// TIA Portal V17 export
// export: Created 2025-05-06T14:32:49.8619923Z, ExportSetting WithDefaults, DisplayName Totally Integrated Automation Portal, DisplayVersion V17 Update 8, DisplayName TIA Portal Openness, DisplayVersion V17 Update 8, DisplayName TIA Portal Version Control Interface, DisplayVersion V17, DisplayName SINAMICS Startdrive Advanced, DisplayVersion V17 SP2, DisplayName SINAMICS Startdrive G110M, G120, G120C, G120D, G120P, G115D, DisplayVersion V17 SP2, DisplayName SINAMICS Startdrive G130, G150, S120, S150, SINAMICS MV, S210, DisplayVersion V17 SP2, DisplayName STEP 7 Professional, DisplayVersion V17 Update 8, DisplayName SINUMERIK ONE STEP 7 Toolbox, DisplayVersion V17 Update 12, DisplayName SINUMERIK 840D sl STEP 7 Toolbox, DisplayVersion V17 Update 12, DisplayName STEP 7 Safety, DisplayVersion V17 Update 6, DisplayName WinCC Advanced, DisplayVersion V17 Update 8
FUNCTION "FC10400_ASPIRATION_PRESSURE_VALUES" : Void   // FC10400, LAD
{ S7_Optimized_Access := 'TRUE' }
VERSION : 0.1
// stored: AutoNumber false, IsIECCheckEnabled false, SetENOAutomatically false, UDAEnableTagReadback false
BEGIN

REGION Network 1: CALL FB10400 PRESSURE SENSOR UNIT 1
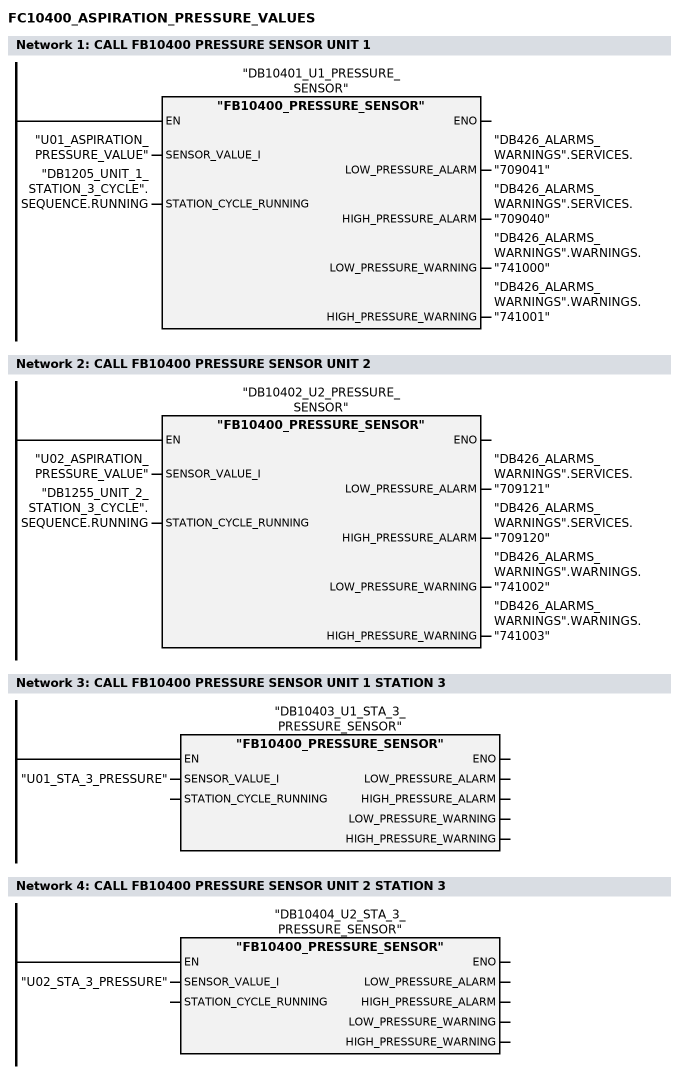
   RUNG wire#powerrail
      "DB10401_U1_PRESSURE_SENSOR"(SENSOR_VALUE_I := "U01_ASPIRATION_PRESSURE_VALUE", STATION_CYCLE_RUNNING := "DB1205_UNIT_1_STATION_3_CYCLE".SEQUENCE.RUNNING, LOW_PRESSURE_ALARM => "DB426_ALARMS_WARNINGS".SERVICES."709041", HIGH_PRESSURE_ALARM => "DB426_ALARMS_WARNINGS".SERVICES."709040", LOW_PRESSURE_WARNING => "DB426_ALARMS_WARNINGS".WARNINGS."741000", HIGH_PRESSURE_WARNING => "DB426_ALARMS_WARNINGS".WARNINGS."741001")
   END_RUNG
   // the same network as SCL:
   "DB10401_U1_PRESSURE_SENSOR"(SENSOR_VALUE_I := "U01_ASPIRATION_PRESSURE_VALUE",   // "FB10400_PRESSURE_SENSOR"
                           STATION_CYCLE_RUNNING := "DB1205_UNIT_1_STATION_3_CYCLE".SEQUENCE.RUNNING,
                           LOW_PRESSURE_ALARM => "DB426_ALARMS_WARNINGS".SERVICES."709041",
                           HIGH_PRESSURE_ALARM => "DB426_ALARMS_WARNINGS".SERVICES."709040",
                           LOW_PRESSURE_WARNING => "DB426_ALARMS_WARNINGS".WARNINGS."741000",
                           HIGH_PRESSURE_WARNING => "DB426_ALARMS_WARNINGS".WARNINGS."741001");
END_REGION

REGION Network 2: CALL FB10400 PRESSURE SENSOR UNIT 2
   RUNG wire#powerrail
      "DB10402_U2_PRESSURE_SENSOR"(SENSOR_VALUE_I := "U02_ASPIRATION_PRESSURE_VALUE", STATION_CYCLE_RUNNING := "DB1255_UNIT_2_STATION_3_CYCLE".SEQUENCE.RUNNING, LOW_PRESSURE_ALARM => "DB426_ALARMS_WARNINGS".SERVICES."709121", HIGH_PRESSURE_ALARM => "DB426_ALARMS_WARNINGS".SERVICES."709120", LOW_PRESSURE_WARNING => "DB426_ALARMS_WARNINGS".WARNINGS."741002", HIGH_PRESSURE_WARNING => "DB426_ALARMS_WARNINGS".WARNINGS."741003")
   END_RUNG
   // the same network as SCL:
   "DB10402_U2_PRESSURE_SENSOR"(SENSOR_VALUE_I := "U02_ASPIRATION_PRESSURE_VALUE",   // "FB10400_PRESSURE_SENSOR"
                           STATION_CYCLE_RUNNING := "DB1255_UNIT_2_STATION_3_CYCLE".SEQUENCE.RUNNING,
                           LOW_PRESSURE_ALARM => "DB426_ALARMS_WARNINGS".SERVICES."709121",
                           HIGH_PRESSURE_ALARM => "DB426_ALARMS_WARNINGS".SERVICES."709120",
                           LOW_PRESSURE_WARNING => "DB426_ALARMS_WARNINGS".WARNINGS."741002",
                           HIGH_PRESSURE_WARNING => "DB426_ALARMS_WARNINGS".WARNINGS."741003");
END_REGION

REGION Network 3: CALL FB10400 PRESSURE SENSOR UNIT 1 STATION 3
   RUNG wire#powerrail
      "DB10403_U1_STA_3_PRESSURE_SENSOR"(SENSOR_VALUE_I := "U01_STA_3_PRESSURE", STATION_CYCLE_RUNNING :=, LOW_PRESSURE_ALARM =>, HIGH_PRESSURE_ALARM =>, LOW_PRESSURE_WARNING =>, HIGH_PRESSURE_WARNING =>)
   END_RUNG
   // the same network as SCL:
   "DB10403_U1_STA_3_PRESSURE_SENSOR"(SENSOR_VALUE_I := "U01_STA_3_PRESSURE");   // "FB10400_PRESSURE_SENSOR"
END_REGION

REGION Network 4: CALL FB10400 PRESSURE SENSOR UNIT 2 STATION 3
   RUNG wire#powerrail
      "DB10404_U2_STA_3_PRESSURE_SENSOR"(SENSOR_VALUE_I := "U02_STA_3_PRESSURE", STATION_CYCLE_RUNNING :=, LOW_PRESSURE_ALARM =>, HIGH_PRESSURE_ALARM =>, LOW_PRESSURE_WARNING =>, HIGH_PRESSURE_WARNING =>)
   END_RUNG
   // the same network as SCL:
   "DB10404_U2_STA_3_PRESSURE_SENSOR"(SENSOR_VALUE_I := "U02_STA_3_PRESSURE");   // "FB10400_PRESSURE_SENSOR"
END_REGION
END_FUNCTION
